# B&R Automation Studio project stocker_muetterlein
Automation Studio 4.5.2.102

## Configuration Config1

CPU X20CP1484-1, AutomationRuntime F3.10, Build 4.1.2, Vc V4.52.0

### Task classes (Cpu.sw)
```
Cyclic#1:
  FSM <- FSM.prg
  PartContro <- PartControl.prg
```

### Hardware
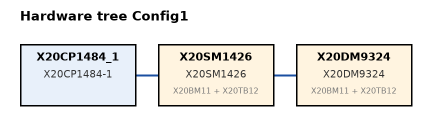
```
X20BM11 : X20BM11 v1.0.0.1  [X2X1 -> X20CP1484_1.IF6]
X20BM11a : X20BM11 v1.0.0.1  [X2X1 -> X20BM11.X2X2]
X20CP1484_1 : X20CP1484-1 v1.1.5.0
  Connector IF2:
    ActivateDevice = 1
    Vnc1
    VncVcObjectName1 = Visu
    VncKeyMappingFile1 = VC\PS2-Keyboard.dis
    VncAuthentication1 = 1
    VncPasswordViewControl1 = abcd
X20DM9324 : X20DM9324 v1.0.4.0  [SS1 -> X20TB12a.SS; SL -> X20BM11a.SL1]
X20SM1426 : X20SM1426 v1.5.1.1  [SS1 -> X20TB12.SS; SL -> X20BM11.SL1]
  FunctionModel = Ramp
  HoldingCurrent01 = 100
  RatedCurrent01 = 100
  MaximumCurrent01 = 100
  MaxSpeed01pos_conf = 2500
  MaxAcc01_conf = 2500
  MaxDec01_conf = 2500
X20TB12 : X20TB12 v1.0.0.0
X20TB12a : X20TB12 v1.0.0.0
```

### IoMap.iom - X20CP1484_1/IoMap.iom
```iecst
VAR_CONFIG
	::DO_LAMP_GREEN AT %QX."X20DM9324".DigitalOutput01;
	::DO_LAMP_RED AT %QX."X20DM9324".DigitalOutput02;
	::DO_PNEO_VENT AT %QX."X20DM9324".DigitalOutput03;
	::DI_SWITCH_GREEN AT %IX."X20DM9324".DigitalInput01;
	::DI_SWITCH_RED AT %IX."X20DM9324".DigitalInput02;
	::DI_LIGHT_SENSE1 AT %IX."X20DM9324".DigitalInput03;
	::AIN_ABS_POS AT %ID."X20SM1426".AbsPos01ActVal;
	::DI_LIGHT_SENSE2  AT %IX."X20DM9324".DigitalInput04;
	::GAI_STATUSWORD AT %IW."X20SM1426".MpGenStatus01;
	::GAO_CONTROLWORD AT %QW."X20SM1426".MpGenControl01;
	::GAO_MOTORMODE AT %QB."X20SM1426".MpGenMode01;
	::GAO_VELOCITY AT %QD."X20SM1426".AbsPos01;
END_VAR
```

## Logical view

### Global.typ - Global data types
```iecst
TYPE
	enumSTATES :
		(
		IDLE := 0,
		STEP1 := 1,
		STEP2 := 2,
		STEP3 := 3
		);
END_TYPE
```

### Global.var - Global variables
```iecst
VAR
	AIN_ABS_POS : DINT;
	aPartLengh : ARRAY[0..29] OF DINT;
	bMotorOn : BOOL := FALSE;
	bWrongSizePartOnPiston : BOOL := FALSE;
	cntParts : UINT := 0;
	cntWaitInput : UINT := 0;
	cntWaitPiston : UINT := 0;
	DI_LIGHT_SENSE1 : BOOL := FALSE;
	DI_LIGHT_SENSE1_OLD : BOOL := FALSE;
	DI_LIGHT_SENSE2 : BOOL := FALSE;
	DI_LIGHT_SENSE2_OLD : BOOL := FALSE;
	DI_SWITCH_GREEN : BOOL := FALSE;
	DI_SWITCH_RED : BOOL := FALSE;
	DO_LAMP_GREEN : BOOL := FALSE;
	DO_LAMP_RED : BOOL := FALSE;
	DO_PNEO_VENT : BOOL := FALSE;
	ENUM_FSM_STATE : enumSTATES := 0;
	idxPartLenghEnd : USINT := 0;
	idxPartLenghStart : USINT := 0;
	PART_LENGH_MAX : {REDUND_UNREPLICABLE} DINT := 120;
	PART_LENGH_MIN : {REDUND_UNREPLICABLE} DINT := 80;
END_VAR
VAR CONSTANT
	SCALE_POS : DINT := 750;
	WAIT_TIME_5S : UINT := 500;
	WAIT_TIME_PISTON : UINT := 200;
END_VAR
VAR
	currentPartStartPos : DINT;
	motor_status : UINT;
	LastPartLengh : DINT := 0;
	GAO_CONTROLWORD : UINT := 0;
	GAO_MOTORMODE : {REDUND_UNREPLICABLE} SINT := 2;
	GAI_STATUSWORD : UINT := 0;
END_VAR
VAR CONSTANT
	GAI_STATUSWORD_MASK : UINT := 15;
END_VAR
VAR
	GAO_VELOCITY : DINT;
	cntPartRej : USINT := 0;
	cntPartOk : USINT := 0;
	LastPartStatus : WSTRING[80];
	cntPartTotal : USINT := 0;
	Velocity : UINT := 1000;
END_VAR
```

### Program Logical/FSM (IEC)

#### Cyclic.st
```iecst
PROGRAM _CYCLIC
	(* Insert code here *)
	CASE ENUM_FSM_STATE OF
		IDLE:
			//check case:
			IF DI_SWITCH_GREEN = TRUE THEN
				//new case:
				ENUM_FSM_STATE := STEP1;
				//set outputs
				DO_LAMP_GREEN := TRUE;
				DO_LAMP_RED := FALSE;
				bMotorOn := TRUE;
			END_IF

		STEP1:
			IF DI_SWITCH_RED = TRUE THEN
				//new case:
				ENUM_FSM_STATE := IDLE;
				//set outputs
				DO_LAMP_GREEN := FALSE;
				DO_LAMP_RED := TRUE;
				bMotorOn := FALSE;
			END_IF
			IF bWrongSizePartOnPiston = TRUE THEN
				//new case:
				ENUM_FSM_STATE := STEP2;
				//set outputs
				bMotorOn := FALSE;
			END_IF
		STEP2:
			cntWaitInput := cntWaitInput -1;
			bWrongSizePartOnPiston := FALSE;
			IF cntWaitInput = 0 THEN //5s timer elapsed = espulsion
				//new case:
				ENUM_FSM_STATE := STEP3;
				//reset counters
				cntWaitInput := WAIT_TIME_5S;
				//set outputs
				DO_PNEO_VENT := 1;
			END_IF
			//check case:
			IF DI_SWITCH_GREEN = TRUE THEN // resume
				//new case:
				ENUM_FSM_STATE := STEP1;
				//reset counters
				cntWaitInput := WAIT_TIME_5S;
				//set outputs
				cntPartOk := cntPartOk + 1;
				bMotorOn := TRUE;
			END_IF

		// here the part is at the piston and will be ejected
		STEP3:
			cntWaitPiston := cntWaitPiston -1;
			IF cntWaitPiston = WAIT_TIME_PISTON / 2 THEN //timer elapsed = espulsion
				DO_PNEO_VENT := 0;
				cntPartRej := cntPartRej+1;
			END_IF
			IF cntWaitPiston = 0 THEN
				//new case:
				ENUM_FSM_STATE := STEP1;
				//reset counters
				cntWaitPiston := WAIT_TIME_PISTON;
				//set outputs
				bMotorOn := TRUE;
			END_IF

	END_CASE
END_PROGRAM
```

#### Exit.st
```iecst
PROGRAM _EXIT
	(* Insert code here *)
END_PROGRAM
```

#### Init.st
```iecst
PROGRAM _INIT
	(* Insert code here *)
	cntWaitInput := WAIT_TIME_5S;
	cntWaitPiston := WAIT_TIME_PISTON;
	ENUM_FSM_STATE := IDLE;
END_PROGRAM
```

### Program Logical/PartControl (IEC)

#### Cyclic.st
```iecst
PROGRAM _CYCLIC
	(* Insert code here *)
	IF ENUM_FSM_STATE = STEP1 THEN
		IF (DI_LIGHT_SENSE1 = TRUE) AND (DI_LIGHT_SENSE1_OLD = FALSE) THEN
			currentPartStartPos := AIN_ABS_POS;
			// TODO ADD velocity
		END_IF
		IF (DI_LIGHT_SENSE1 = FALSE) AND (DI_LIGHT_SENSE1_OLD = TRUE) THEN
			LastPartLengh := (AIN_ABS_POS - currentPartStartPos) / SCALE_POS;
			aPartLengh[idxPartLenghStart] := LastPartLengh;
			cntParts := cntParts +1;
			//add to queue:
			IF idxPartLenghStart >19 THEN
				idxPartLenghStart := 0;
			ELSE
				idxPartLenghStart := idxPartLenghStart +1;
			END_IF
		END_IF

		IF (DI_LIGHT_SENSE2 = TRUE) AND (DI_LIGHT_SENSE2_OLD = FALSE) THEN
			cntPartTotal := cntPartTotal + 1;
			IF (aPartLengh[idxPartLenghEnd] <= PART_LENGH_MIN) THEN
				bWrongSizePartOnPiston := TRUE;
				LastPartStatus := "TOO SHORT";
			ELSIF (aPartLengh[idxPartLenghEnd] >= PART_LENGH_MAX) THEN
				bWrongSizePartOnPiston := TRUE;
				LastPartStatus := "TOO LONG";
			ELSE
				cntPartOk := cntPartOk + 1;
				LastPartStatus := "OK";
			END_IF
		END_IF

	END_IF

	IF (DI_LIGHT_SENSE2 = FALSE) AND (DI_LIGHT_SENSE2_OLD = TRUE) THEN
		IF idxPartLenghEnd >19 THEN
			idxPartLenghEnd := 0;
		ELSE
			idxPartLenghEnd := idxPartLenghEnd +1;
		END_IF
		cntParts := cntParts - 1;
	END_IF

	DI_LIGHT_SENSE1_OLD := DI_LIGHT_SENSE1;
	DI_LIGHT_SENSE2_OLD := DI_LIGHT_SENSE2;

END_PROGRAM
```

- Visualisation Logical/Visu (not shown)

### Program Logical/MotorControl (IEC)

#### Cyclic.st
```iecst
PROGRAM _CYCLIC
	(* Insert code here *)
	motor_status := (GAI_STATUSWORD AND GAI_STATUSWORD_MASK);
	IF motor_status = 7 THEN 			// STATUS_OPERATION_ENABLED
		IF bMotorOn = TRUE THEN
			GAO_VELOCITY := Velocity;
		ELSE
			GAO_VELOCITY := 0;
		END_IF
	ELSIF motor_status = 3 THEN		//STATUS_SWITCHED_ON
		GAO_CONTROLWORD := 15;		//CONTROL_OPERATION_ENABLED
	ELSIF motor_status = 1 THEN	//Status_READY_TO_SWITCH_ON
		GAO_CONTROLWORD := 7;		// CONTROL_SWITCH_ON
	ELSE
		GAO_CONTROLWORD := 6;		// CONTROL_SHUTDOWN
	END_IF

END_PROGRAM
```

#### Init.st
```iecst
PROGRAM _INIT
	(* Insert code here *)
	GAO_MOTORMODE := 2;
END_PROGRAM
```

Listed in the project but not available here: Logical/Libraries
